// TwinCAT 3 PLC project EventLogger
// ProgramVersion: 3.1.4023.0
// libraries:
//   Tc2_Standard, * (Beckhoff Automation GmbH)
//   Tc2_System, * (Beckhoff Automation GmbH)
//   Tc2_Utilities, * (Beckhoff Automation GmbH)
//   Tc3_Module, * (Beckhoff Automation GmbH)
// project tree:
//   DUTs/ E_Type.TcDUT, ST_Event.TcDUT
//   / PlcTask.TcTTO
//   POUs/ FB_CSVEventStorage.TcPOU, FB_EventLogger.TcPOU, F_EventTimeStamp.TcPOU, I_CSVEventStorage.TcIO, MAIN.TcPOU

CONFIGURATION EventLogger
    RESOURCE PLC ON TwinCAT3
        TASK PlcTask(INTERVAL := T#10ms, PRIORITY := 20);
        PROGRAM MAIN WITH PlcTask : MAIN;
    END_RESOURCE
END_CONFIGURATION

// ---- DUTs/E_Type.TcDUT
{attribute 'qualified_only'}
{attribute 'strict'}
{attribute 'to_string'}
TYPE E_Type :
(
	alarm := 0,
	message := 1
);
END_TYPE

// ---- DUTs/ST_Event.TcDUT
TYPE ST_Event :
STRUCT
	eEventType : E_Type;
	eEventSeverity : TCEventSeverity;
	nEventDefinition : UINT;
	sEventMessage : STRING(255);
	tTimeStamp : DATE_AND_TIME;	
END_STRUCT
END_TYPE

// ---- POUs/I_CSVEventStorage.TcIO
INTERFACE I_CSVEventStorage

METHOD StoreEvent
VAR_INPUT
	stEvent : ST_Event;
END_VAR
END_METHOD

END_INTERFACE

// ---- POUs/MAIN.TcPOU
PROGRAM MAIN
VAR	
	//Test event
	stEvent : ST_Event;	
	bAddEvent : BOOL;
	CSVEventStorage : FB_CSVEventStorage;	
	fbEventLogger : FB_EventLogger(CSVEventStorage);
END_VAR

//Assign event values
stEvent.eEventType := E_Type.alarm;
stEvent.eEventSeverity := TCEventSeverity.Critical;
stEvent.nEventDefinition := 30;
stEvent.sEventMessage := 'Something went wrong';

//Run only once to add an event
IF bAddEvent THEN
	fbEventLogger.AddEvent(stEvent);
	bAddEvent := FALSE;
END_IF

END_PROGRAM

// ---- POUs/FB_CSVEventStorage.TcPOU
FUNCTION_BLOCK FB_CSVEventStorage IMPLEMENTS I_CSVEventStorage
VAR_INPUT
END_VAR
VAR_OUTPUT
END_VAR
VAR
END_VAR

{warning 'add method implementation '}
METHOD StoreEvent
VAR_INPUT
	stEvent	: ST_Event;
END_VAR
END_METHOD

END_FUNCTION_BLOCK

// ---- POUs/FB_EventLogger.TcPOU
FUNCTION_BLOCK FB_EventLogger
VAR
	aEventBuffer : ARRAY[1..nBufferSize] OF ST_Event;
	nBufferIndex : INT := 0;
	_iCSVEventStorage : I_CSVEventStorage;	
END_VAR

VAR CONSTANT
	nBufferSize : INT := 50;
END_VAR

METHOD PUBLIC AddEvent : BOOL
VAR_IN_OUT
	stEvent : ST_Event;
END_VAR
IF NOT CheckEventBuffer() THEN
	nBufferIndex := nBufferIndex + 1;
	aEventBuffer[nBufferIndex].eEventType := stEvent.eEventType;
	aEventBuffer[nBufferIndex].eEventSeverity:= stEvent.eEventSeverity;
	aEventBuffer[nBufferIndex].nEventDefinition := stEvent.nEventDefinition;
	aEventBuffer[nBufferIndex].sEventMessage := stEvent.sEventMessage;
	F_EventTimeStamp(aEventBuffer[nBufferIndex]);
	AddEvent := TRUE;	
ELSE
	AddEvent := FALSE; 
END_IF

//Store event in the CSV file
_iCSVEventStorage.StoreEvent(stEvent := aEventBuffer[nBufferIndex]);
END_METHOD

(*Returns True if event buffer full, False otherwise*)
METHOD PRIVATE CheckEventBuffer : BOOL
VAR_INPUT
END_VAR
IF (nBufferIndex + 1 > nBufferSize) THEN
	CheckEventBuffer := TRUE;
ELSE
	CheckEventBuffer := FALSE;
END_IF
END_METHOD

METHOD FB_init : BOOL
VAR_INPUT
	bInitRetains : BOOL; // if TRUE, the retain variables are initialized (warm start / cold start)
	bInCopyCode : BOOL;  // if TRUE, the instance afterwards gets moved into the copy code (online change)
	iCSVEventStorage : I_CSVEventStorage;
END_VAR
_iCSVEventStorage := iCSVEventStorage;
END_METHOD

END_FUNCTION_BLOCK

// ---- POUs/F_EventTimeStamp.TcPOU
FUNCTION F_EventTimeStamp
VAR_IN_OUT
	stEvent : ST_Event;
END_VAR
VAR
	stFileTime : T_FILETIME;
	fbGetSystemTime : GETSYSTEMTIME;
END_VAR

fbGetSystemTime(timeLoDW => stFileTime.dwLowDateTime, timeHiDW => stfiletime.dwHighDateTime);
stEvent.tTimeStamp := FileTime_To_Dt(filetime := stFileTime);

END_FUNCTION
